{attribute 'qualified_only'}
VAR_GLOBAL CONSTANT
	MaxAmountManagers				: UINT := 10;
END_VAR

(* stored: Version 1.1.0.1
   GVL Par_Manager: Id {24cac663-fc0c-46a3-9043-5bebd1146c9a}, ParameterList True *)
